FUNCTION_BLOCK TelemetryRelativeHumiditiesWidget 
VAR_INPUT
END_VAR
VAR_OUTPUT
END_VAR
VAR_IN_OUT
    ref : TelemetryRelativeHumidities;
END_VAR
VAR
    actualStatus : StatusWidget;
    // temperatures
    topAir                  : MeasurementWidget('Top air', '%.1f %%');
    insideTube              : MeasurementWidget('Inside tube', '%.2f %%');
END_VAR

actualStatus(text := ref.actualStatus, color := HealthToColor(ref.statuses.healthStatus));

_update(ref.topAir, topAir);
_update(ref.insideTube, insideTube);

METHOD _update : BOOL
VAR_INPUT
END_VAR
VAR_IN_OUT
    ref : RelativeHumidityMeasurement;
    widget : MeasurementWidget;
END_VAR
widget(
    value        := ref.average.percent.value, 
    actualStatus := ref.actualStatus,
    healthStatus := ref.statuses.healthStatus);
END_METHOD

END_FUNCTION_BLOCK

(* stored: Version 1.1.0.1, ProductVersion 3.1.4018.2
   POU TelemetryRelativeHumiditiesWidget: Id {0e603c46-6a54-40de-a666-5d3dc09f0222}, SpecialFunc None
   Method _update: Id {f37938e7-b740-4d5b-89fa-2881c80f8af4} *)
